FUNCTION_BLOCK CompositeBlockWithoutConnections
  FBS
    BaseBlock1 : BaseBlock;
    EA_2_router : EA_2_router;
    EA_network1 : EA_network1;
    EA_network1_2 : EA_network1;
    EA_LeftPublishSubscribeAdapter : EA_LeftPublishSubscribeAdapter;
    Publish_Left_EA : PUBLISH_5;
    Subscribe_Left_EA : SUBSCRIBE_5;
    EA_LeftPublishSubscribeAdapter_2 : EA_LeftPublishSubscribeAdapter;
    Publish_Left_EA_2 : PUBLISH_5;
    Subscribe_Left_EA_2 : SUBSCRIBE_5;
  END_FBS
  EVENT_CONNECTIONS
    EA_LeftPublishSubscribeAdapter.REQ TO Publish_Left_EA.REQ;
    Subscribe_Left_EA.IND TO EA_LeftPublishSubscribeAdapter.IND;
    EA_LeftPublishSubscribeAdapter_2.REQ TO Publish_Left_EA_2.REQ;
    Subscribe_Left_EA_2.IND TO EA_LeftPublishSubscribeAdapter_2.IND;
  END_CONNECTIONS
  DATA_CONNECTIONS
    EA_LeftPublishSubscribeAdapter.I_E_number TO Publish_Left_EA.SD_1;
    EA_LeftPublishSubscribeAdapter.O_data1 TO Publish_Left_EA.SD_2;
    EA_LeftPublishSubscribeAdapter.O_data2 TO Publish_Left_EA.SD_3;
    EA_LeftPublishSubscribeAdapter.N_I_data1 TO Publish_Left_EA.SD_4;
    EA_LeftPublishSubscribeAdapter.N_I_data2 TO Publish_Left_EA.SD_5;
    Subscribe_Left_EA.RD_1 TO EA_LeftPublishSubscribeAdapter.O_E_number;
    Subscribe_Left_EA.RD_2 TO EA_LeftPublishSubscribeAdapter.I_data1;
    Subscribe_Left_EA.RD_3 TO EA_LeftPublishSubscribeAdapter.I_data2;
    Subscribe_Left_EA.RD_4 TO EA_LeftPublishSubscribeAdapter.N_O_data1;
    Subscribe_Left_EA.RD_5 TO EA_LeftPublishSubscribeAdapter.N_O_data2;
    EA_LeftPublishSubscribeAdapter_2.I_E_number TO Publish_Left_EA_2.SD_1;
    EA_LeftPublishSubscribeAdapter_2.O_data1 TO Publish_Left_EA_2.SD_2;
    EA_LeftPublishSubscribeAdapter_2.O_data2 TO Publish_Left_EA_2.SD_3;
    EA_LeftPublishSubscribeAdapter_2.N_I_data1 TO Publish_Left_EA_2.SD_4;
    EA_LeftPublishSubscribeAdapter_2.N_I_data2 TO Publish_Left_EA_2.SD_5;
    Subscribe_Left_EA_2.RD_1 TO EA_LeftPublishSubscribeAdapter_2.O_E_number;
    Subscribe_Left_EA_2.RD_2 TO EA_LeftPublishSubscribeAdapter_2.I_data1;
    Subscribe_Left_EA_2.RD_3 TO EA_LeftPublishSubscribeAdapter_2.I_data2;
    Subscribe_Left_EA_2.RD_4 TO EA_LeftPublishSubscribeAdapter_2.N_O_data1;
    Subscribe_Left_EA_2.RD_5 TO EA_LeftPublishSubscribeAdapter_2.N_O_data2;
  END_CONNECTIONS
  ADAPTER_CONNECTIONS
    BaseBlock1.plug TO EA_2_router.socket;
    EA_2_router.plug_0 TO EA_network1.socket;
    EA_2_router.plug_1 TO EA_network1_2.socket;
    EA_network1.plug TO EA_LeftPublishSubscribeAdapter.socket;
    EA_network1_2.plug TO EA_LeftPublishSubscribeAdapter_2.socket;
  END_CONNECTIONS
END_FUNCTION_BLOCK
